INTERFACE I_RpcResponseManagerConfig

END_INTERFACE

(* stored: Version 1.1.0.1, ProductVersion 3.1.4024.12
   Itf I_RpcResponseManagerConfig: Id {4a4f0798-ed83-499b-b5a8-20a54d5c473a} *)
